PROGRAM main
VAR
	Lid_at_place AT %IX100.0 : bool; (* pokrywka przed zaciskiem *)
	Lid_clamped AT %IX100.1 : bool;
	Base_at_place AT %IX100.2 : bool;
	Base_clamped AT %IX100.3 : bool;
	Moving_X AT %IX100.4 : bool;
	Moving_Z AT %IX100.5 : bool;
	Item_detected AT %IX100.6 : bool; (* Grabbed sucesfully *)
	Part_leaving AT %IX100.7 : bool;
	Lids_conveyor AT %QX100.0 : bool;
	Clamp_lid AT %QX100.1 : bool; (* zacisnij *)
	Pos_raise_lid AT %QX100.2 : bool;
	Base_conveyor AT %QX100.3 : bool;
	Clamp_base AT %QX100.4 : bool;
	Move_X AT %QX100.5 : bool;
	Move_Z AT %QX100.6 : bool;
	Grab AT %QX100.7 : bool;
	Start AT %IX101.0 : bool;
	Delay : time := T#500ms;
	TON0 : TON;
	TOF0 : TOF;
	TOF1 : TOF;
	TON3 : TON;
	TOF2 : TON;
END_VAR

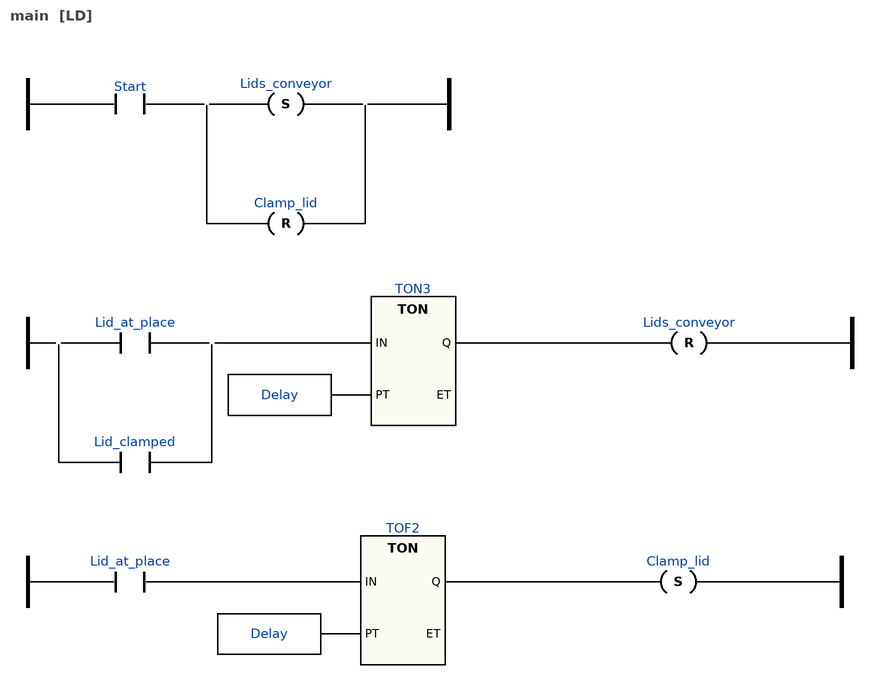
(* LD diagram, written out as Structured Text *)
IF Start THEN Lids_conveyor := TRUE; END_IF;
IF Start THEN Clamp_lid := FALSE; END_IF;
TON3(IN := Lid_at_place OR Lid_clamped, PT := Delay);
IF TON3.Q THEN Lids_conveyor := FALSE; END_IF;
TOF2(IN := Lid_at_place, PT := Delay);
IF TOF2.Q THEN Clamp_lid := TRUE; END_IF;
END_PROGRAM
